// TIA Portal V19 export
FUNCTION_BLOCK "A0303_Spintore_FB"   // FB80, LAD
TITLE = GESTIONE SPINTORE
// stored: MemoryReserve 100, SetENOAutomatically false
   VAR_INPUT
      AreaInterface : "AreaInterface";
      ZSI : "udt_ZoneSafetyInterface";
      DSI : "udt_DeviceSafetyInterface";
      DataIn : Struct
         OP_Rest_PB : Bool;
         OP_Work_PB : Bool;
         LsPosition1 : Bool;   // FTC CONTROLLO PEZZO IN 1 POSIZIONE STRATO
         LsMaxPosition : Bool;   // FTC CONTROLLO MASSIMA POSIZIONE 1=ALLARME
      END_STRUCT;
      CIn : Struct
         Manager : Struct
            EnableStopDoorOpeningReq : Bool;
            EnableStopInPhase : Bool;
            EnableStopProgrammed : Bool;
            Control_ON : Bool;
            CanMoveFreely : Bool;
            Rest : Bool;
            Work : Bool;
         END_STRUCT;
         Manip : Struct
            OutOfWorkspace : Bool;
         END_STRUCT;
      END_STRUCT;
      Config : Struct
         Testa : Struct
            Vrt : "ValveMachine_Config";
            Orz : "ValveMachine_Config";
         END_STRUCT;
         Coda : Struct
            Vrt : "ValveMachine_Config";
            Orz : "ValveMachine_Config";
         END_STRUCT;
         DelayMissingCondition { ExternalAccessible := 'False'; ExternalVisible := 'False'; ExternalWritable := 'False'} : Time := T#0MS;
      END_STRUCT;
   END_VAR
   VAR_OUTPUT
      MachineInterface : "MachineInterface";
      COut : Struct
         Vrt : "ValveMachine_COut";
         Orz : "ValveMachine_COut";
      END_STRUCT;
   END_VAR
   VAR
      Alarm : Struct
         Testa : Struct
            Vrt : "ValveAlr";
            Orz : "ValveAlr";
         END_STRUCT;
         Coda : Struct
            Vrt : "ValveAlr";
            Orz : "ValveAlr";
         END_STRUCT;
         PassaggioPezzoNonOK : Bool;
      END_STRUCT;
      Warning : Struct
         Testa : Struct
            Vrt : "ValveMachine_Wng";
            Orz : "ValveMachine_Wng";
         END_STRUCT;
         Coda : Struct
            Vrt : "ValveMachine_Wng";
            Orz : "ValveMachine_Wng";
         END_STRUCT;
         OP_REST_MissingCnd : Bool;   // Mancanza comando arresto
         OP_WORK_MissingCnd : Bool;   // Mancanza consenso lavoro
      END_STRUCT;
      HMI : Struct
         Selection : Struct
            Vrt : Int;   // 0= BOTH ; 1= HEAD ; 2= TAIL
            Orz : Int;   // 0= BOTH ; 1= HEAD ; 2= TAIL
         END_STRUCT;
      END_STRUCT;
      Ctrl : Struct
         OP_Rest_Man : Bool;
         OP_Work_Man : Bool;
         OP_Rest_Aut : Bool;
         OP_Work_Aut : Bool;
         OP_Rest : Bool;
         OP_Work : Bool;
      END_STRUCT;
      Sts : Struct
         OP_Ax_CanMoveFreely : Bool;
         OP_Rest_Cnd : Bool;
         OP_Work_Cnd : Bool;
      END_STRUCT;
      Vrt_Testa : "ValveMachine_FB";
      Vrt_Coda : "ValveMachine_FB";
      Orz_Testa : "ValveMachine_FB";
      Orz_Coda : "ValveMachine_FB";
      AUX : Struct
         OP_Rest_PB { ExternalAccessible := 'False'; ExternalVisible := 'False'; ExternalWritable := 'False'} : Bool;
         OP_Work_PB { ExternalAccessible := 'False'; ExternalVisible := 'False'; ExternalWritable := 'False'} : Bool;
         LsPosition1_PE { ExternalAccessible := 'False'; ExternalVisible := 'False'; ExternalWritable := 'False'} : Bool;
         LsPosition1_NE { ExternalAccessible := 'False'; ExternalVisible := 'False'; ExternalWritable := 'False'} : Bool;
      END_STRUCT;
      TON_OP_REST_MissingCnd : IEC_TIMER;
      TON_OP_WORK_MissingCnd : IEC_TIMER;
      TON_CheckPos1Ok { S7_SetPoint := 'True'} : IEC_TIMER;
   END_VAR
   VAR_TEMP
      PE : Struct
         OP_Rest_PB : Bool;
         OP_Work_PB : Bool;
         LsPosition1 : Bool;
      END_STRUCT;
      NE : Struct
         LsPosition1 : Bool;
      END_STRUCT;
      i : Int;
   END_VAR
   // Config.Testa.Vrt.DelayPressureRunningTimeout := T#3S;
   // Config.Testa.Vrt.DelayMissingCondition := T#3S;
   // Config.Testa.Vrt.Rest_LsQty := 1;
   // Config.Testa.Vrt.Work_LsQty := 1;
   // Config.Testa.Vrt.Rest_RetainAut := FALSE;
   // Config.Testa.Vrt.Work_RetainAut := FALSE;
   // Config.Testa.Vrt.V.RestLimSwitchExist := TRUE;
   // Config.Testa.Vrt.V.WorkLimSwitchExist := TRUE;
   // Config.Testa.Vrt.V.CheckOilInPressure := FALSE;
   // Config.Testa.Vrt.V.CutRestWhenIsAtRest := TRUE;
   // Config.Testa.Vrt.V.CutWorkWhenIsAtWork := TRUE;
   // Config.Testa.Vrt.V.RestTime := T#0MS;
   // Config.Testa.Vrt.V.WorkTime := T#0MS;
   // Config.Testa.Vrt.V.RestTimeOut := T#2S;
   // Config.Testa.Vrt.V.WorkTimeOut := T#2S;
   // Config.Testa.Orz.DelayPressureRunningTimeout := T#3S;
   // Config.Testa.Orz.DelayMissingCondition := T#3S;
   // Config.Testa.Orz.Rest_LsQty := 1;
   // Config.Testa.Orz.Work_LsQty := 1;
   // Config.Testa.Orz.Rest_RetainAut := FALSE;
   // Config.Testa.Orz.Work_RetainAut := FALSE;
   // Config.Testa.Orz.V.RestLimSwitchExist := TRUE;
   // Config.Testa.Orz.V.WorkLimSwitchExist := TRUE;
   // Config.Testa.Orz.V.CheckOilInPressure := FALSE;
   // Config.Testa.Orz.V.CutRestWhenIsAtRest := TRUE;
   // Config.Testa.Orz.V.CutWorkWhenIsAtWork := TRUE;
   // Config.Testa.Orz.V.RestTime := T#0MS;
   // Config.Testa.Orz.V.WorkTime := T#0MS;
   // Config.Testa.Orz.V.RestTimeOut := T#2S;
   // Config.Testa.Orz.V.WorkTimeOut := T#2S;
   // Config.Coda.Vrt.DelayPressureRunningTimeout := T#3S;
   // Config.Coda.Vrt.DelayMissingCondition := T#3S;
   // Config.Coda.Vrt.Rest_LsQty := 1;
   // Config.Coda.Vrt.Work_LsQty := 1;
   // Config.Coda.Vrt.Rest_RetainAut := FALSE;
   // Config.Coda.Vrt.Work_RetainAut := FALSE;
   // Config.Coda.Vrt.V.RestLimSwitchExist := TRUE;
   // Config.Coda.Vrt.V.WorkLimSwitchExist := TRUE;
   // Config.Coda.Vrt.V.CheckOilInPressure := FALSE;
   // Config.Coda.Vrt.V.CutRestWhenIsAtRest := TRUE;
   // Config.Coda.Vrt.V.CutWorkWhenIsAtWork := TRUE;
   // Config.Coda.Vrt.V.RestTime := T#0MS;
   // Config.Coda.Vrt.V.WorkTime := T#0MS;
   // Config.Coda.Vrt.V.RestTimeOut := T#2S;
   // Config.Coda.Vrt.V.WorkTimeOut := T#2S;
   // Config.Coda.Orz.DelayPressureRunningTimeout := T#3S;
   // Config.Coda.Orz.DelayMissingCondition := T#3S;
   // Config.Coda.Orz.Rest_LsQty := 1;
   // Config.Coda.Orz.Work_LsQty := 1;
   // Config.Coda.Orz.Rest_RetainAut := FALSE;
   // Config.Coda.Orz.Work_RetainAut := FALSE;
   // Config.Coda.Orz.V.RestLimSwitchExist := TRUE;
   // Config.Coda.Orz.V.WorkLimSwitchExist := TRUE;
   // Config.Coda.Orz.V.CheckOilInPressure := FALSE;
   // Config.Coda.Orz.V.CutRestWhenIsAtRest := TRUE;
   // Config.Coda.Orz.V.CutWorkWhenIsAtWork := TRUE;
   // Config.Coda.Orz.V.RestTime := T#0MS;
   // Config.Coda.Orz.V.WorkTime := T#0MS;
   // Config.Coda.Orz.V.RestTimeOut := T#2S;
   // Config.Coda.Orz.V.WorkTimeOut := T#2S;
   VAR_TEMP   // added for the SCL form of the ladder/FBD networks
      _w1 : Bool;
      _w2 : Bool;
      _w3 : Bool;
   END_VAR
BEGIN

REGION Network 1 (SCL): Reset allarmi
   IF #AreaInterface.RstAlarms THEN
       ;
   END_IF;
END_REGION

REGION Network 2: <+>
END_REGION

REGION Network 3: Fronti Sensori
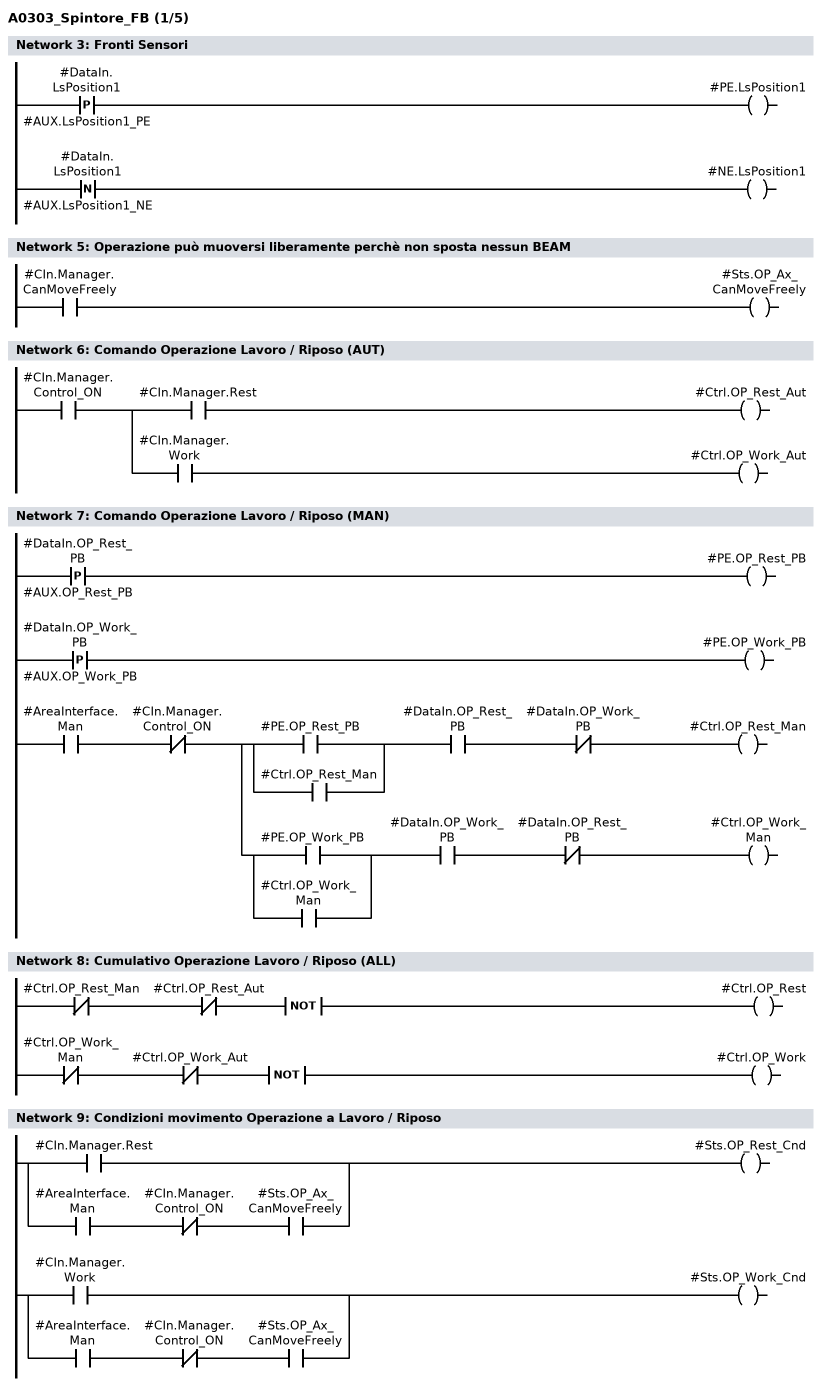
   RUNG wire#powerrail
      P_Contact(operand := #DataIn.LsPosition1, bit := #AUX.LsPosition1_PE)
      Coil( #PE.LsPosition1 )
   END_RUNG
   RUNG wire#powerrail
      N_Contact(operand := #DataIn.LsPosition1, bit := #AUX.LsPosition1_NE)
      Coil( #NE.LsPosition1 )
   END_RUNG
   // the same network as SCL:
   #_w1 := #DataIn.LsPosition1 AND NOT #AUX.LsPosition1_PE;   // rising edge of #DataIn.LsPosition1
   #AUX.LsPosition1_PE := #DataIn.LsPosition1;
   #PE.LsPosition1 := #_w1;
   #_w2 := NOT #DataIn.LsPosition1 AND #AUX.LsPosition1_NE;   // falling edge of #DataIn.LsPosition1
   #AUX.LsPosition1_NE := #DataIn.LsPosition1;
   #NE.LsPosition1 := #_w2;
END_REGION

REGION Network 4: <+>
END_REGION

REGION Network 5: Operazione può muoversi liberamente perchè non sposta nessun BEAM
   RUNG wire#powerrail
      Contact( #CIn.Manager.CanMoveFreely )
      Coil( #Sts.OP_Ax_CanMoveFreely )
   END_RUNG
   // the same network as SCL:
   #Sts.OP_Ax_CanMoveFreely := #CIn.Manager.CanMoveFreely;
END_REGION

REGION Network 6: Comando Operazione Lavoro / Riposo (AUT)
   RUNG wire#powerrail
      Contact( #CIn.Manager.Control_ON )
      wire#w1
      Contact( #CIn.Manager.Rest )
      Coil( #Ctrl.OP_Rest_Aut )
   END_RUNG
   RUNG wire#w1
      Contact( #CIn.Manager.Work )
      Coil( #Ctrl.OP_Work_Aut )
   END_RUNG
   // the same network as SCL:
   #Ctrl.OP_Rest_Aut := #CIn.Manager.Control_ON AND #CIn.Manager.Rest;
   #Ctrl.OP_Work_Aut := #CIn.Manager.Control_ON AND #CIn.Manager.Work;
END_REGION

REGION Network 7: Comando Operazione Lavoro / Riposo (MAN)
   RUNG wire#powerrail
      P_Contact(operand := #DataIn.OP_Rest_PB, bit := #AUX.OP_Rest_PB)
      Coil( #PE.OP_Rest_PB )
   END_RUNG
   RUNG wire#powerrail
      P_Contact(operand := #DataIn.OP_Work_PB, bit := #AUX.OP_Work_PB)
      Coil( #PE.OP_Work_PB )
   END_RUNG
   RUNG wire#powerrail
      Contact( #AreaInterface.Man )
      I_Contact( #CIn.Manager.Control_ON )
      wire#w1
      Contact( #PE.OP_Rest_PB )
      wire#w2
      Contact( #DataIn.OP_Rest_PB )
      I_Contact( #DataIn.OP_Work_PB )
      Coil( #Ctrl.OP_Rest_Man )
   END_RUNG
   RUNG wire#w1
      Contact( #Ctrl.OP_Rest_Man )
   END_RUNG wire#w2
   RUNG wire#w1
      Contact( #PE.OP_Work_PB )
      wire#w3
      Contact( #DataIn.OP_Work_PB )
      I_Contact( #DataIn.OP_Rest_PB )
      Coil( #Ctrl.OP_Work_Man )
   END_RUNG
   RUNG wire#w1
      Contact( #Ctrl.OP_Work_Man )
   END_RUNG wire#w3
   // the same network as SCL:
   #_w1 := #DataIn.OP_Rest_PB AND NOT #AUX.OP_Rest_PB;   // rising edge of #DataIn.OP_Rest_PB
   #AUX.OP_Rest_PB := #DataIn.OP_Rest_PB;
   #PE.OP_Rest_PB := #_w1;
   #_w2 := #DataIn.OP_Work_PB AND NOT #AUX.OP_Work_PB;   // rising edge of #DataIn.OP_Work_PB
   #AUX.OP_Work_PB := #DataIn.OP_Work_PB;
   #PE.OP_Work_PB := #_w2;
   #_w3 := #AreaInterface.Man AND NOT #CIn.Manager.Control_ON;
   #Ctrl.OP_Rest_Man := #_w3 AND (#PE.OP_Rest_PB OR #Ctrl.OP_Rest_Man) AND #DataIn.OP_Rest_PB AND NOT #DataIn.OP_Work_PB;
   #Ctrl.OP_Work_Man := #_w3 AND (#PE.OP_Work_PB OR #Ctrl.OP_Work_Man) AND #DataIn.OP_Work_PB AND NOT #DataIn.OP_Rest_PB;
END_REGION

REGION Network 8: Cumulativo Operazione Lavoro / Riposo (ALL)
   RUNG wire#powerrail
      I_Contact( #Ctrl.OP_Rest_Man )
      I_Contact( #Ctrl.OP_Rest_Aut )
      Not()
      Coil( #Ctrl.OP_Rest )
   END_RUNG
   RUNG wire#powerrail
      I_Contact( #Ctrl.OP_Work_Man )
      I_Contact( #Ctrl.OP_Work_Aut )
      Not()
      Coil( #Ctrl.OP_Work )
   END_RUNG
   // the same network as SCL:
   #Ctrl.OP_Rest := NOT (NOT #Ctrl.OP_Rest_Man AND NOT #Ctrl.OP_Rest_Aut);
   #Ctrl.OP_Work := NOT (NOT #Ctrl.OP_Work_Man AND NOT #Ctrl.OP_Work_Aut);
END_REGION

REGION Network 9: Condizioni movimento Operazione a Lavoro / Riposo
   RUNG wire#powerrail
      Contact( #CIn.Manager.Rest )
      wire#w1
      Coil( #Sts.OP_Rest_Cnd )
   END_RUNG
   RUNG wire#powerrail
      Contact( #AreaInterface.Man )
      I_Contact( #CIn.Manager.Control_ON )
      Contact( #Sts.OP_Ax_CanMoveFreely )
   END_RUNG wire#w1
   RUNG wire#powerrail
      Contact( #CIn.Manager.Work )
      wire#w2
      Coil( #Sts.OP_Work_Cnd )
   END_RUNG
   RUNG wire#powerrail
      Contact( #AreaInterface.Man )
      I_Contact( #CIn.Manager.Control_ON )
      Contact( #Sts.OP_Ax_CanMoveFreely )
   END_RUNG wire#w2
   // the same network as SCL:
   #Sts.OP_Rest_Cnd := #CIn.Manager.Rest OR (#AreaInterface.Man AND NOT #CIn.Manager.Control_ON AND #Sts.OP_Ax_CanMoveFreely);
   #Sts.OP_Work_Cnd := #CIn.Manager.Work OR (#AreaInterface.Man AND NOT #CIn.Manager.Control_ON AND #Sts.OP_Ax_CanMoveFreely);
END_REGION

REGION Network 10: <+>
END_REGION

REGION Network 11 (SCL): Verticale + Orizzontale - Cin Manager (Esecuzione sequenza comandi)
   #Vrt_Testa.Cin.Manager.Control_ON := #Vrt_Coda.Cin.Manager.Control_ON :=
   #Orz_Testa.Cin.Manager.Control_ON := #Orz_Coda.Cin.Manager.Control_ON := #Ctrl.OP_Rest OR #Ctrl.OP_Work;
   //
   #Vrt_Testa.Cin.Manager.Rest := FALSE;
   #Vrt_Coda.Cin.Manager.Rest := FALSE;
   #Orz_Testa.Cin.Manager.Rest := FALSE;
   #Orz_Coda.Cin.Manager.Rest := FALSE;

   //************************************
   #Vrt_Testa.Cin.Manager.Work := FALSE;
   #Vrt_Coda.Cin.Manager.Work:= FALSE;
   #Orz_Testa.Cin.Manager.Work := FALSE;
   #Orz_Coda.Cin.Manager.Work := FALSE;
   //

   IF #Ctrl.OP_Rest AND #Sts.OP_Rest_Cnd THEN

       #Vrt_Testa.Cin.Manager.Rest := NOT #Vrt_Testa.COut.Rest;
       #Vrt_Coda.Cin.Manager.Rest := NOT #Vrt_Coda.COut.Rest;
       #Orz_Testa.Cin.Manager.Rest := #Vrt_Testa.COut.Rest AND #Vrt_Coda.COut.Rest;
       #Orz_Coda.Cin.Manager.Rest := #Vrt_Testa.COut.Rest AND #Vrt_Coda.COut.Rest;


   ELSIF #Ctrl.OP_Work AND #Sts.OP_Work_Cnd THEN


       #Vrt_Testa.Cin.Manager.Work := #Orz_Testa.COut.Rest;
       #Vrt_Coda.Cin.Manager.Work := #Orz_Coda.COut.Rest;

       #Orz_Testa.Cin.Manager.Work := #Vrt_Testa.COut.Work AND #Vrt_Coda.COut.Work;
       #Orz_Coda.Cin.Manager.Work := #Vrt_Testa.COut.Work AND #Vrt_Coda.COut.Work;



   END_IF;
END_REGION

REGION Network 12 (SCL): Verticale + Orizzontale - CIn Abilitazioni Manager
   //Stop Door Opening Request
   #Vrt_Testa.Cin.Manager.EnableStopDoorOpeningReq := #Vrt_Coda.Cin.Manager.EnableStopDoorOpeningReq :=
   #Orz_Testa.Cin.Manager.EnableStopDoorOpeningReq := #Orz_Coda.Cin.Manager.EnableStopDoorOpeningReq := #CIn.Manager.EnableStopDoorOpeningReq;

   //Stop In Phase
   #Vrt_Testa.Cin.Manager.EnableStopInPhase := #Vrt_Coda.Cin.Manager.EnableStopInPhase :=
   #Orz_Testa.Cin.Manager.EnableStopInPhase := #Orz_Coda.Cin.Manager.EnableStopInPhase := #CIn.Manager.EnableStopInPhase;

   //Stop Programmed
   #Vrt_Testa.Cin.Manager.EnableStopProgrammed := #Vrt_Coda.Cin.Manager.EnableStopProgrammed :=
   #Orz_Testa.Cin.Manager.EnableStopProgrammed := #Orz_Coda.Cin.Manager.EnableStopProgrammed := #CIn.Manager.EnableStopProgrammed;
END_REGION

REGION Network 13: <+>
END_REGION

REGION Network 14: Warning manacanza condizioni esecuzione Operazione RIPOSO / LAVORO
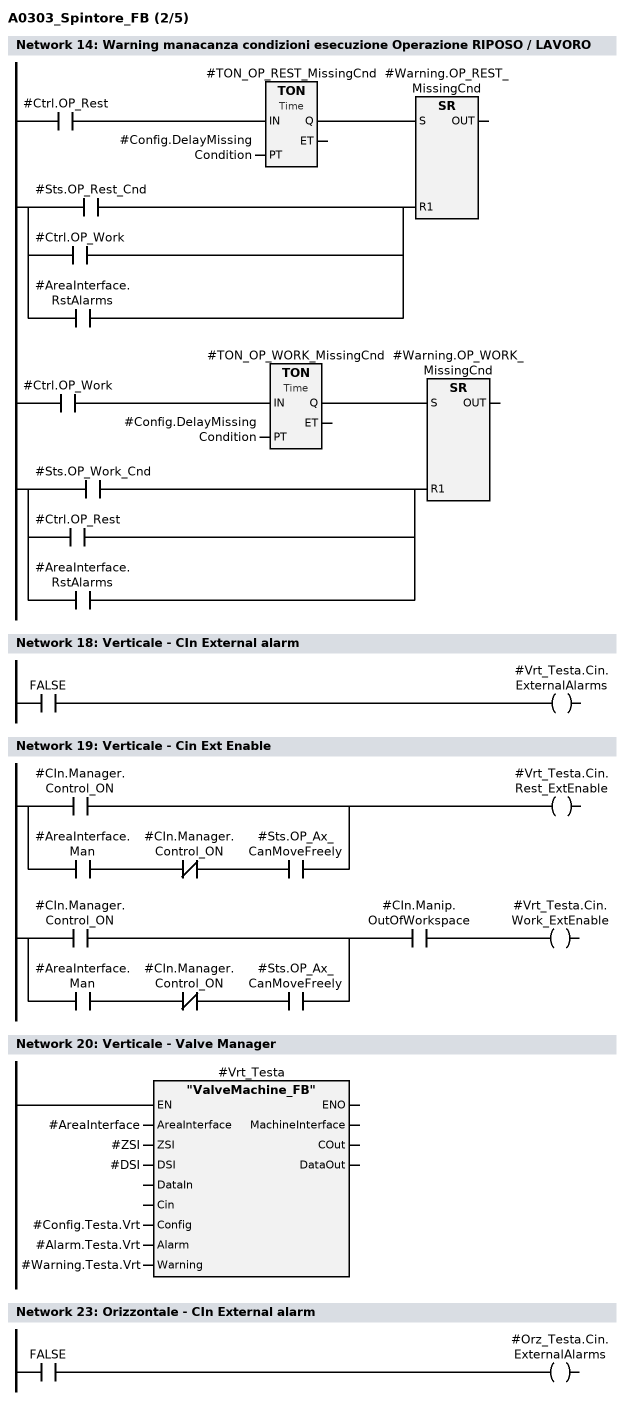
   RUNG wire#powerrail
      Contact( #Ctrl.OP_Rest )
      { S7_Templates := "time_type := Time" } #TON_OP_REST_MissingCnd.TON(pt := #Config.DelayMissingCondition, et =>)
      S_SR(operand := #Warning.OP_REST_MissingCnd, r1 := wire#w1)
   END_RUNG
   RUNG wire#powerrail
      Contact( #Sts.OP_Rest_Cnd )
   END_RUNG wire#w1
   RUNG wire#powerrail
      Contact( #Ctrl.OP_Work )
   END_RUNG wire#w1
   RUNG wire#powerrail
      Contact( #AreaInterface.RstAlarms )
   END_RUNG wire#w1
   RUNG wire#powerrail
      Contact( #Ctrl.OP_Work )
      { S7_Templates := "time_type := Time" } #TON_OP_WORK_MissingCnd.TON(pt := #Config.DelayMissingCondition, et =>)
      S_SR(operand := #Warning.OP_WORK_MissingCnd, r1 := wire#w2)
   END_RUNG
   RUNG wire#powerrail
      Contact( #Sts.OP_Work_Cnd )
   END_RUNG wire#w2
   RUNG wire#powerrail
      Contact( #Ctrl.OP_Rest )
   END_RUNG wire#w2
   RUNG wire#powerrail
      Contact( #AreaInterface.RstAlarms )
   END_RUNG wire#w2
   // the same network as SCL:
   #TON_OP_REST_MissingCnd.TON(IN := #Ctrl.OP_Rest, PT := #Config.DelayMissingCondition);
   IF #TON_OP_REST_MissingCnd.Q THEN
       #Warning.OP_REST_MissingCnd := TRUE;   // SR flip-flop
   END_IF;
   IF #Sts.OP_Rest_Cnd OR #Ctrl.OP_Work OR #AreaInterface.RstAlarms THEN
       #Warning.OP_REST_MissingCnd := FALSE;
   END_IF;
   #TON_OP_WORK_MissingCnd.TON(IN := #Ctrl.OP_Work, PT := #Config.DelayMissingCondition);
   IF #TON_OP_WORK_MissingCnd.Q THEN
       #Warning.OP_WORK_MissingCnd := TRUE;   // SR flip-flop
   END_IF;
   IF #Sts.OP_Work_Cnd OR #Ctrl.OP_Rest OR #AreaInterface.RstAlarms THEN
       #Warning.OP_WORK_MissingCnd := FALSE;
   END_IF;
END_REGION

REGION Network 15: <+>
END_REGION

REGION Network 16: <<<<<<<<<<<<<<<<<<<<<<<<< LATO TESTA >>>>>>>>>>>>>>>>>>>>>>>>>>>>>>>>>>>>>>>>>
END_REGION

REGION Network 17: << GESTIONE VERTICALE >>
END_REGION

REGION Network 18: Verticale - CIn External alarm
   RUNG wire#powerrail
      Contact( FALSE )
      Coil( #Vrt_Testa.Cin.ExternalAlarms )
   END_RUNG
   // the same network as SCL:
   #Vrt_Testa.Cin.ExternalAlarms := FALSE;
END_REGION

REGION Network 19: Verticale - Cin Ext Enable
   RUNG wire#powerrail
      Contact( #CIn.Manager.Control_ON )
      wire#w1
      Coil( #Vrt_Testa.Cin.Rest_ExtEnable )
   END_RUNG
   RUNG wire#powerrail
      Contact( #AreaInterface.Man )
      I_Contact( #CIn.Manager.Control_ON )
      Contact( #Sts.OP_Ax_CanMoveFreely )
   END_RUNG wire#w1
   RUNG wire#powerrail
      Contact( #CIn.Manager.Control_ON )
      wire#w2
      Contact( #CIn.Manip.OutOfWorkspace )
      Coil( #Vrt_Testa.Cin.Work_ExtEnable )
   END_RUNG
   RUNG wire#powerrail
      Contact( #AreaInterface.Man )
      I_Contact( #CIn.Manager.Control_ON )
      Contact( #Sts.OP_Ax_CanMoveFreely )
   END_RUNG wire#w2
   // the same network as SCL:
   #Vrt_Testa.Cin.Rest_ExtEnable := #CIn.Manager.Control_ON OR (#AreaInterface.Man AND NOT #CIn.Manager.Control_ON AND #Sts.OP_Ax_CanMoveFreely);
   #Vrt_Testa.Cin.Work_ExtEnable := (#CIn.Manager.Control_ON OR (#AreaInterface.Man AND NOT #CIn.Manager.Control_ON AND #Sts.OP_Ax_CanMoveFreely)) AND #CIn.Manip.OutOfWorkspace;
END_REGION

REGION Network 20: Verticale - Valve Manager
   RUNG wire#powerrail
      #Vrt_Testa(AreaInterface := #AreaInterface, ZSI := #ZSI, DSI := #DSI, DataIn :=, Cin :=, Config := #Config.Testa.Vrt, Alarm := #Alarm.Testa.Vrt, Warning := #Warning.Testa.Vrt, MachineInterface =>, COut =>, DataOut =>)
   END_RUNG
   // the same network as SCL:
   #Vrt_Testa(AreaInterface := #AreaInterface,   // "ValveMachine_FB"
              ZSI := #ZSI,
              DSI := #DSI,
              Config := #Config.Testa.Vrt,
              Alarm := #Alarm.Testa.Vrt,
              Warning := #Warning.Testa.Vrt);
END_REGION

REGION Network 21: <+>
END_REGION

REGION Network 22: << GESTIONE ORIZZONTALE >>
END_REGION

REGION Network 23: Orizzontale - CIn External alarm
   RUNG wire#powerrail
      Contact( FALSE )
      Coil( #Orz_Testa.Cin.ExternalAlarms )
   END_RUNG
   // the same network as SCL:
   #Orz_Testa.Cin.ExternalAlarms := FALSE;
END_REGION

REGION Network 24: Orizzontale - Cin Ext Enable
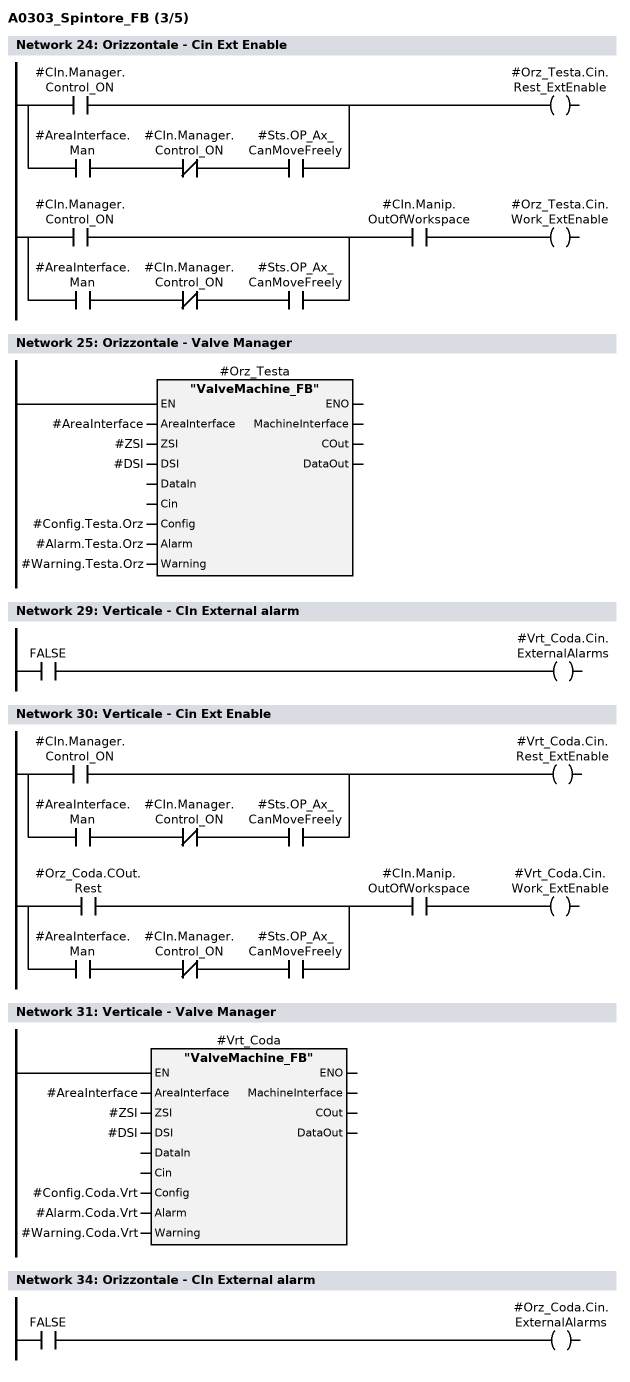
   RUNG wire#powerrail
      Contact( #CIn.Manager.Control_ON )
      wire#w1
      Coil( #Orz_Testa.Cin.Rest_ExtEnable )
   END_RUNG
   RUNG wire#powerrail
      Contact( #AreaInterface.Man )
      I_Contact( #CIn.Manager.Control_ON )
      Contact( #Sts.OP_Ax_CanMoveFreely )
   END_RUNG wire#w1
   RUNG wire#powerrail
      Contact( #CIn.Manager.Control_ON )
      wire#w2
      Contact( #CIn.Manip.OutOfWorkspace )
      Coil( #Orz_Testa.Cin.Work_ExtEnable )
   END_RUNG
   RUNG wire#powerrail
      Contact( #AreaInterface.Man )
      I_Contact( #CIn.Manager.Control_ON )
      Contact( #Sts.OP_Ax_CanMoveFreely )
   END_RUNG wire#w2
   // the same network as SCL:
   #Orz_Testa.Cin.Rest_ExtEnable := #CIn.Manager.Control_ON OR (#AreaInterface.Man AND NOT #CIn.Manager.Control_ON AND #Sts.OP_Ax_CanMoveFreely);
   #Orz_Testa.Cin.Work_ExtEnable := (#CIn.Manager.Control_ON OR (#AreaInterface.Man AND NOT #CIn.Manager.Control_ON AND #Sts.OP_Ax_CanMoveFreely)) AND #CIn.Manip.OutOfWorkspace;
END_REGION

REGION Network 25: Orizzontale - Valve Manager
   RUNG wire#powerrail
      #Orz_Testa(AreaInterface := #AreaInterface, ZSI := #ZSI, DSI := #DSI, DataIn :=, Cin :=, Config := #Config.Testa.Orz, Alarm := #Alarm.Testa.Orz, Warning := #Warning.Testa.Orz, MachineInterface =>, COut =>, DataOut =>)
   END_RUNG
   // the same network as SCL:
   #Orz_Testa(AreaInterface := #AreaInterface,   // "ValveMachine_FB"
              ZSI := #ZSI,
              DSI := #DSI,
              Config := #Config.Testa.Orz,
              Alarm := #Alarm.Testa.Orz,
              Warning := #Warning.Testa.Orz);
END_REGION

REGION Network 26: <+>
END_REGION

REGION Network 27: <<<<<<<<<<<<<<<<<<<<<<<<< LATO CODA >>>>>>>>>>>>>>>>>>>>>>>>>>>>>>>>>>>>>>>>>
END_REGION

REGION Network 28: << GESTIONE VERTICALE >>
END_REGION

REGION Network 29: Verticale - CIn External alarm
   RUNG wire#powerrail
      Contact( FALSE )
      Coil( #Vrt_Coda.Cin.ExternalAlarms )
   END_RUNG
   // the same network as SCL:
   #Vrt_Coda.Cin.ExternalAlarms := FALSE;
END_REGION

REGION Network 30: Verticale - Cin Ext Enable
   RUNG wire#powerrail
      Contact( #CIn.Manager.Control_ON )
      wire#w1
      Coil( #Vrt_Coda.Cin.Rest_ExtEnable )
   END_RUNG
   RUNG wire#powerrail
      Contact( #AreaInterface.Man )
      I_Contact( #CIn.Manager.Control_ON )
      Contact( #Sts.OP_Ax_CanMoveFreely )
   END_RUNG wire#w1
   RUNG wire#powerrail
      Contact( #Orz_Coda.COut.Rest )
      wire#w2
      Contact( #CIn.Manip.OutOfWorkspace )
      Coil( #Vrt_Coda.Cin.Work_ExtEnable )
   END_RUNG
   RUNG wire#powerrail
      Contact( #AreaInterface.Man )
      I_Contact( #CIn.Manager.Control_ON )
      Contact( #Sts.OP_Ax_CanMoveFreely )
   END_RUNG wire#w2
   // the same network as SCL:
   #Vrt_Coda.Cin.Rest_ExtEnable := #CIn.Manager.Control_ON OR (#AreaInterface.Man AND NOT #CIn.Manager.Control_ON AND #Sts.OP_Ax_CanMoveFreely);
   #Vrt_Coda.Cin.Work_ExtEnable := (#Orz_Coda.COut.Rest OR (#AreaInterface.Man AND NOT #CIn.Manager.Control_ON AND #Sts.OP_Ax_CanMoveFreely)) AND #CIn.Manip.OutOfWorkspace;
END_REGION

REGION Network 31: Verticale - Valve Manager
   RUNG wire#powerrail
      #Vrt_Coda(AreaInterface := #AreaInterface, ZSI := #ZSI, DSI := #DSI, DataIn :=, Cin :=, Config := #Config.Coda.Vrt, Alarm := #Alarm.Coda.Vrt, Warning := #Warning.Coda.Vrt, MachineInterface =>, COut =>, DataOut =>)
   END_RUNG
   // the same network as SCL:
   #Vrt_Coda(AreaInterface := #AreaInterface,   // "ValveMachine_FB"
             ZSI := #ZSI,
             DSI := #DSI,
             Config := #Config.Coda.Vrt,
             Alarm := #Alarm.Coda.Vrt,
             Warning := #Warning.Coda.Vrt);
END_REGION

REGION Network 32: <+>
END_REGION

REGION Network 33: << GESTIONE ORIZZONTALE >>
END_REGION

REGION Network 34: Orizzontale - CIn External alarm
   RUNG wire#powerrail
      Contact( FALSE )
      Coil( #Orz_Coda.Cin.ExternalAlarms )
   END_RUNG
   // the same network as SCL:
   #Orz_Coda.Cin.ExternalAlarms := FALSE;
END_REGION

REGION Network 35: Orizzontale - Cin Ext Enable
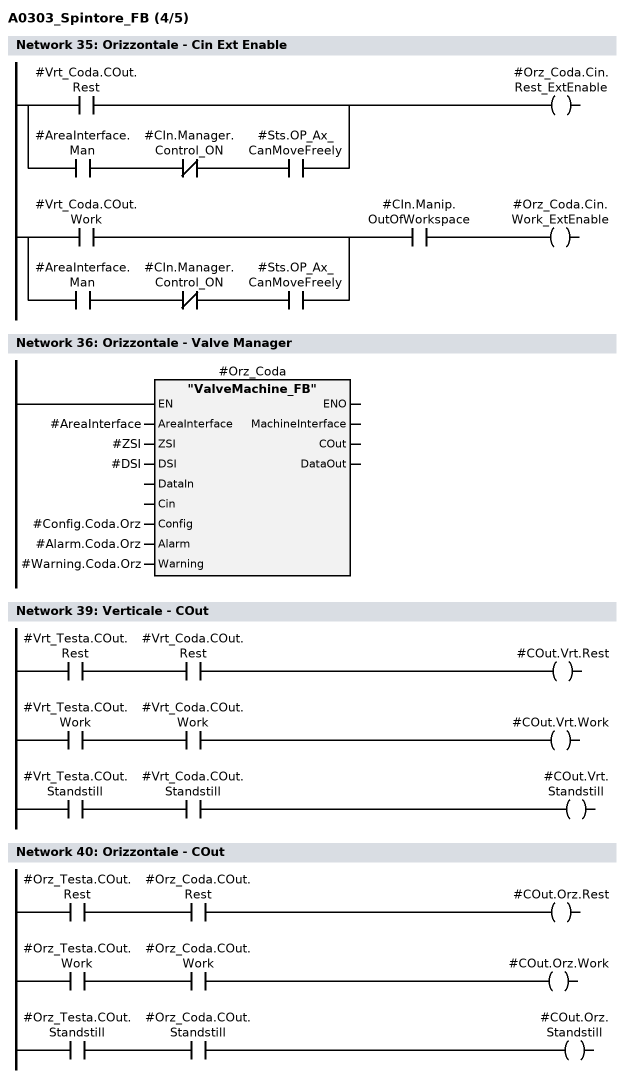
   RUNG wire#powerrail
      Contact( #Vrt_Coda.COut.Rest )
      wire#w1
      Coil( #Orz_Coda.Cin.Rest_ExtEnable )
   END_RUNG
   RUNG wire#powerrail
      Contact( #AreaInterface.Man )
      I_Contact( #CIn.Manager.Control_ON )
      Contact( #Sts.OP_Ax_CanMoveFreely )
   END_RUNG wire#w1
   RUNG wire#powerrail
      Contact( #Vrt_Coda.COut.Work )
      wire#w2
      Contact( #CIn.Manip.OutOfWorkspace )
      Coil( #Orz_Coda.Cin.Work_ExtEnable )
   END_RUNG
   RUNG wire#powerrail
      Contact( #AreaInterface.Man )
      I_Contact( #CIn.Manager.Control_ON )
      Contact( #Sts.OP_Ax_CanMoveFreely )
   END_RUNG wire#w2
   // the same network as SCL:
   #Orz_Coda.Cin.Rest_ExtEnable := #Vrt_Coda.COut.Rest OR (#AreaInterface.Man AND NOT #CIn.Manager.Control_ON AND #Sts.OP_Ax_CanMoveFreely);
   #Orz_Coda.Cin.Work_ExtEnable := (#Vrt_Coda.COut.Work OR (#AreaInterface.Man AND NOT #CIn.Manager.Control_ON AND #Sts.OP_Ax_CanMoveFreely)) AND #CIn.Manip.OutOfWorkspace;
END_REGION

REGION Network 36: Orizzontale - Valve Manager
   RUNG wire#powerrail
      #Orz_Coda(AreaInterface := #AreaInterface, ZSI := #ZSI, DSI := #DSI, DataIn :=, Cin :=, Config := #Config.Coda.Orz, Alarm := #Alarm.Coda.Orz, Warning := #Warning.Coda.Orz, MachineInterface =>, COut =>, DataOut =>)
   END_RUNG
   // the same network as SCL:
   #Orz_Coda(AreaInterface := #AreaInterface,   // "ValveMachine_FB"
             ZSI := #ZSI,
             DSI := #DSI,
             Config := #Config.Coda.Orz,
             Alarm := #Alarm.Coda.Orz,
             Warning := #Warning.Coda.Orz);
END_REGION

REGION Network 37: <+>
END_REGION

REGION Network 38: <<< COut >>>
END_REGION

REGION Network 39: Verticale - COut
   RUNG wire#powerrail
      Contact( #Vrt_Testa.COut.Rest )
      Contact( #Vrt_Coda.COut.Rest )
      Coil( #COut.Vrt.Rest )
   END_RUNG
   RUNG wire#powerrail
      Contact( #Vrt_Testa.COut.Work )
      Contact( #Vrt_Coda.COut.Work )
      Coil( #COut.Vrt.Work )
   END_RUNG
   RUNG wire#powerrail
      Contact( #Vrt_Testa.COut.Standstill )
      Contact( #Vrt_Coda.COut.Standstill )
      Coil( #COut.Vrt.Standstill )
   END_RUNG
   // the same network as SCL:
   #COut.Vrt.Rest := #Vrt_Testa.COut.Rest AND #Vrt_Coda.COut.Rest;
   #COut.Vrt.Work := #Vrt_Testa.COut.Work AND #Vrt_Coda.COut.Work;
   #COut.Vrt.Standstill := #Vrt_Testa.COut.Standstill AND #Vrt_Coda.COut.Standstill;
END_REGION

REGION Network 40: Orizzontale - COut
   RUNG wire#powerrail
      Contact( #Orz_Testa.COut.Rest )
      Contact( #Orz_Coda.COut.Rest )
      Coil( #COut.Orz.Rest )
   END_RUNG
   RUNG wire#powerrail
      Contact( #Orz_Testa.COut.Work )
      Contact( #Orz_Coda.COut.Work )
      Coil( #COut.Orz.Work )
   END_RUNG
   RUNG wire#powerrail
      Contact( #Orz_Testa.COut.Standstill )
      Contact( #Orz_Coda.COut.Standstill )
      Coil( #COut.Orz.Standstill )
   END_RUNG
   // the same network as SCL:
   #COut.Orz.Rest := #Orz_Testa.COut.Rest AND #Orz_Coda.COut.Rest;
   #COut.Orz.Work := #Orz_Testa.COut.Work AND #Orz_Coda.COut.Work;
   #COut.Orz.Standstill := #Orz_Testa.COut.Standstill AND #Orz_Coda.COut.Standstill;
END_REGION

REGION Network 42: <<< MACHINE STATUS >>>
END_REGION

REGION Network 43: Collect machine to zone interface (internal machines OR)
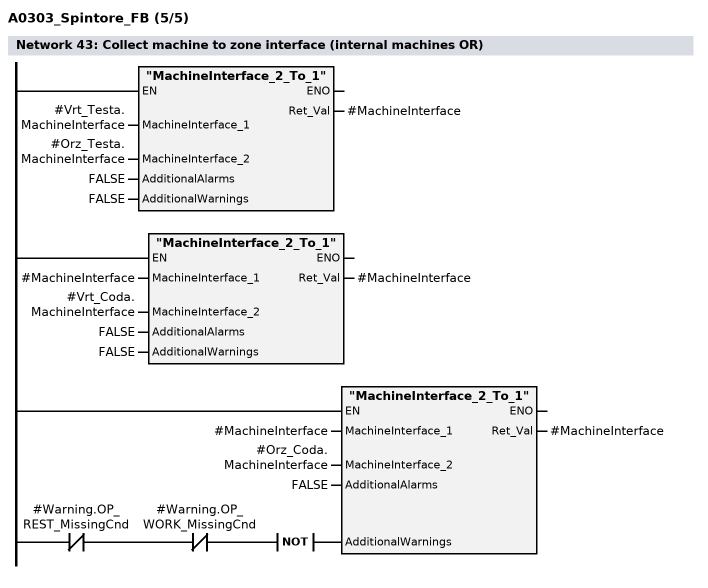
   RUNG wire#powerrail
      "MachineInterface_2_To_1"(MachineInterface_1 := #Vrt_Testa.MachineInterface, MachineInterface_2 := #Orz_Testa.MachineInterface, AdditionalAlarms := FALSE, AdditionalWarnings := FALSE, Ret_Val => #MachineInterface)
   END_RUNG
   RUNG wire#powerrail
      "MachineInterface_2_To_1"(MachineInterface_1 := #MachineInterface, MachineInterface_2 := #Vrt_Coda.MachineInterface, AdditionalAlarms := FALSE, AdditionalWarnings := FALSE, Ret_Val => #MachineInterface)
   END_RUNG
   RUNG wire#powerrail
      "MachineInterface_2_To_1"(AdditionalWarnings := wire#w1, MachineInterface_1 := #MachineInterface, MachineInterface_2 := #Orz_Coda.MachineInterface, AdditionalAlarms := FALSE, Ret_Val => #MachineInterface)
   END_RUNG
   RUNG wire#powerrail
      I_Contact( #Warning.OP_REST_MissingCnd )
      I_Contact( #Warning.OP_WORK_MissingCnd )
      Not()
   END_RUNG wire#w1
   // the same network as SCL:
   #MachineInterface := "MachineInterface_2_To_1"(MachineInterface_1 := #Vrt_Testa.MachineInterface,
                           MachineInterface_2 := #Orz_Testa.MachineInterface,
                           AdditionalAlarms := FALSE,
                           AdditionalWarnings := FALSE);
   #MachineInterface := "MachineInterface_2_To_1"(MachineInterface_1 := #MachineInterface,
                           MachineInterface_2 := #Vrt_Coda.MachineInterface,
                           AdditionalAlarms := FALSE,
                           AdditionalWarnings := FALSE);
   #MachineInterface := "MachineInterface_2_To_1"(MachineInterface_1 := #MachineInterface,
                           MachineInterface_2 := #Orz_Coda.MachineInterface,
                           AdditionalAlarms := FALSE,
                           AdditionalWarnings := NOT (NOT #Warning.OP_REST_MissingCnd AND NOT #Warning.OP_WORK_MissingCnd));
END_REGION
END_FUNCTION_BLOCK
